ABB RobotStudio station: Solution_20200504-211433.rsstn

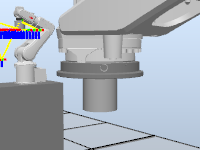
Station Solution (saved by RobotStudio 7.0.8743.626)
Controller Controller
  mechanical unit ROB_1: IRB120_3_58__01, 6 joints, base frame (-200, 0, 800) mm
  mechanical unit ROB_2: IRB120_3_58__01_2, 6 joints, base frame (200, 0, 800) mm, rotated rx 0 ry 0 rz 180 deg
  mechanical unit ROB_3: IRB760_450_318__01, 6 joints, base frame (0, 4000, 0) mm
Layout (positions relative to the parent item):
  - IRB120_3_58__01 [mechanism, from Robots\IRB120_3_58_G_01.rslib] at (-200, 0, 800) mm; joint values [0, -0.7948, 0.351, 0, 2.0145, 0] (rad or m)
  - IRB120_3_58__01_2 [mechanism, from Robots\IRB120_3_58_G_01.rslib] at (200, 0, 800) mm, rotated rx 0 ry 0 rz 180 deg; joint values [0, -0.7948, 0.351, 0, 2.0145, 0] (rad or m)
  - IRB760_450_318__01 [mechanism, from Robots\IRB760_450_318__01.rslib] at (0, 4000, 0) mm; joint values [-1.1097, -0.0075, 0.5664, -1.1097] (rad or m)
  - Part_1 [part]
  - Tool_1 [mechanism] at (-150, 0, 1400) mm, rotated rx 180 ry 0 rz 180 deg
      TCP Tool1 at (0, 0, 0) mm
      links: SimpleGripper
  - Tool_2 [mechanism] at (150, 0, 1400) mm, rotated rx 180 ry 0 rz 0 deg
      TCP Tool_2 at (0, 0, 0) mm
      links: SimpleGripper
  - Tool_3 [mechanism] at (765, 2460, 1100) mm, rotated rx 180 ry 0 rz 180 deg
      TCP Tool_3 at (0, 0, 0) mm
      links: SimpleGripper
Attachment: Tool_1 is attached to IRB120_3_58__01 / Link6
Attachment: Tool_2 is attached to IRB120_3_58__01_2 / Link6
Attachment: Tool_3 is attached to IRB760_450_318__01 / Link6
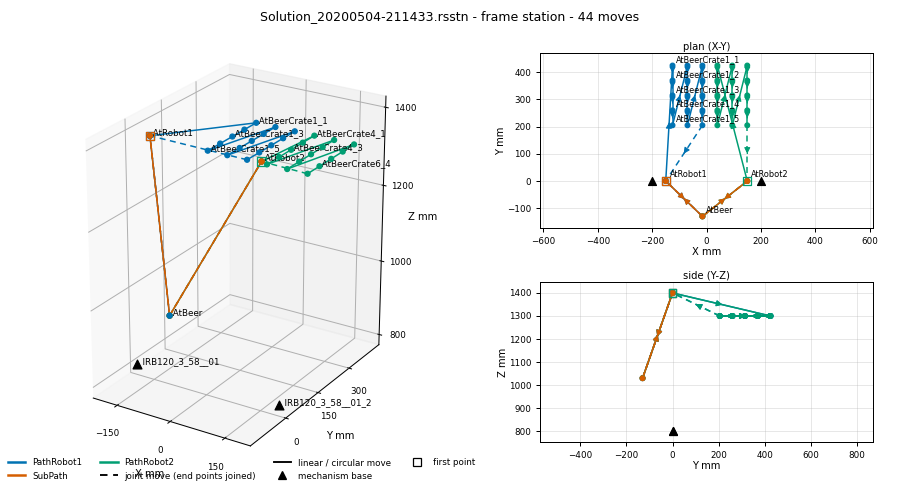
[picture p0: tool path of Solution_20200504-211433.rsstn in frame station, 44 of 44 moves have a stored position in this frame; points joined in program order, loops and branches not executed]
Targets, tools, work objects and paths stored in the station, written as RAPID:
! task T_ROB1
MODULE CalibData
  PERS tooldata Tool1:=[TRUE,[[0,0,0],[1,0,0,0]],[1,[0,0,1],[1,0,0,0],0,0,0]];
ENDMODULE

! task T_ROB1
MODULE Module1
  CONST robtarget AtBeer:=[[-15,-130,1030],[0,0,1,0],[-1,0,-1,0],[9E+09,9E+09,9E+09,9E+09,9E+09,9E+09]];
  CONST robtarget AtRobot1:=[[-150,0,1400],[0,0,1,0],[0,0,0,0],[9E+09,9E+09,9E+09,9E+09,9E+09,9E+09]];
  CONST robtarget AtBeerCrate1_1:=[[-125,425,1300],[0,0,1,0],[0,0,0,0],[9E+09,9E+09,9E+09,9E+09,9E+09,9E+09]];
  CONST robtarget AtBeerCrate1_2:=[[-125,370,1300],[0,0,1,0],[0,0,0,0],[9E+09,9E+09,9E+09,9E+09,9E+09,9E+09]];
  CONST robtarget AtBeerCrate1_3:=[[-125,315,1300],[0,0,1,0],[0,0,0,0],[9E+09,9E+09,9E+09,9E+09,9E+09,9E+09]];
  CONST robtarget AtBeerCrate1_4:=[[-125,260,1300],[0,0,1,0],[0,0,0,0],[9E+09,9E+09,9E+09,9E+09,9E+09,9E+09]];
  CONST robtarget AtBeerCrate1_5:=[[-125,205,1300],[0,0,1,0],[0,0,0,0],[9E+09,9E+09,9E+09,9E+09,9E+09,9E+09]];
  CONST robtarget AtBeerCrate2_1:=[[-70,425,1300],[0,0,1,0],[0,0,0,0],[9E+09,9E+09,9E+09,9E+09,9E+09,9E+09]];
  CONST robtarget AtBeerCrate2_2:=[[-70,370,1300],[0,0,1,0],[0,0,0,0],[9E+09,9E+09,9E+09,9E+09,9E+09,9E+09]];
  CONST robtarget AtBeerCrate2_3:=[[-70,315,1300],[0,0,1,0],[0,0,0,0],[9E+09,9E+09,9E+09,9E+09,9E+09,9E+09]];
  CONST robtarget AtBeerCrate2_4:=[[-70,260,1300],[0,0,1,0],[0,0,0,0],[9E+09,9E+09,9E+09,9E+09,9E+09,9E+09]];
  CONST robtarget AtBeerCrate2_5:=[[-70,205,1300],[0,0,1,0],[0,0,0,0],[9E+09,9E+09,9E+09,9E+09,9E+09,9E+09]];
  CONST robtarget AtBeerCrate3_1:=[[-15,425,1300],[0,0,1,0],[0,0,0,0],[9E+09,9E+09,9E+09,9E+09,9E+09,9E+09]];
  CONST robtarget AtBeerCrate3_2:=[[-15,370,1300],[0,0,1,0],[0,0,0,0],[9E+09,9E+09,9E+09,9E+09,9E+09,9E+09]];
  CONST robtarget AtBeerCrate3_3:=[[-15,315,1300],[0,0,1,0],[0,0,0,0],[9E+09,9E+09,9E+09,9E+09,9E+09,9E+09]];
  CONST robtarget AtBeerCrate3_4:=[[-15,260,1300],[0,0,1,0],[0,0,0,0],[9E+09,9E+09,9E+09,9E+09,9E+09,9E+09]];
  CONST robtarget AtBeerCrate3_5:=[[-15,205,1300],[0,0,1,0],[0,0,0,0],[9E+09,9E+09,9E+09,9E+09,9E+09,9E+09]];
  PROC main()
    PathRobot1;
  ENDPROC
  PROC PathRobot1()
    MoveJ AtRobot1,v2000,z100,Tool1\WObj:=wobj0;
    MoveL AtBeer,v2000,fine,Tool1\WObj:=wobj0;
    SetDO Do1Gripper,1;
    WaitTime 0.3;
    MoveJ AtRobot1,v2000,z100,Tool1\WObj:=wobj0;
    MoveL AtBeerCrate1_1,v2000,fine,Tool1\WObj:=wobj0;
    SubPath;
    MoveL AtBeerCrate1_2,v2000,fine,Tool1\WObj:=wobj0;
    SubPath;
    MoveL AtBeerCrate1_3,v2000,fine,Tool1\WObj:=wobj0;
    SubPath;
    MoveL AtBeerCrate1_4,v2000,fine,Tool1\WObj:=wobj0;
    SubPath;
    MoveL AtBeerCrate1_5,v2000,fine,Tool1\WObj:=wobj0;
    SubPath;
    MoveL AtBeerCrate2_1,v2000,fine,Tool1\WObj:=wobj0;
    SubPath;
    MoveL AtBeerCrate2_2,v2000,fine,Tool1\WObj:=wobj0;
    SubPath;
    MoveL AtBeerCrate2_3,v2000,fine,Tool1\WObj:=wobj0;
    SubPath;
    MoveL AtBeerCrate2_4,v2000,fine,Tool1\WObj:=wobj0;
    SubPath;
    MoveL AtBeerCrate2_5,v2000,fine,Tool1\WObj:=wobj0;
    SubPath;
    MoveL AtBeerCrate3_1,v2000,fine,Tool1\WObj:=wobj0;
    SubPath;
    MoveL AtBeerCrate3_2,v2000,fine,Tool1\WObj:=wobj0;
    SubPath;
    MoveL AtBeerCrate3_3,v2000,fine,Tool1\WObj:=wobj0;
    SubPath;
    MoveL AtBeerCrate3_4,v2000,fine,Tool1\WObj:=wobj0;
    SubPath;
    MoveL AtBeerCrate3_5,v2000,fine,Tool1\WObj:=wobj0;
    SetDO Do1Gripper,0;
    WaitTime 0.3;
    MoveJ AtRobot1,v2000,z100,Tool1\WObj:=wobj0;
  ENDPROC
  PROC SubPath()
    SetDO Do1Gripper,0;
    WaitTime 0.3;
    MoveJ AtRobot1,v2000,z100,Tool1\WObj:=wobj0;
    MoveL AtBeer,v2000,fine,Tool1\WObj:=wobj0;
    SetDO Do1Gripper,1;
    WaitTime 0.3;
    MoveJ AtRobot1,v2000,z100,Tool1\WObj:=wobj0;
  ENDPROC
ENDMODULE

! task T_ROB2
MODULE Module1
  CONST robtarget AtBeer:=[[-15,-130,1030],[0,1,0,0],[0,0,0,0],[9E+09,9E+09,9E+09,9E+09,9E+09,9E+09]];
  CONST robtarget AtRobot2:=[[150,0,1400],[0,1,0,0],[0,0,0,0],[9E+09,9E+09,9E+09,9E+09,9E+09,9E+09]];
  CONST robtarget AtBeerCrate4_1:=[[40,425,1300],[0,1,0,0],[-1,0,-1,0],[9E+09,9E+09,9E+09,9E+09,9E+09,9E+09]];
  CONST robtarget AtBeerCrate4_2:=[[40,370,1300],[0,1,0,0],[-1,0,-1,0],[9E+09,9E+09,9E+09,9E+09,9E+09,9E+09]];
  CONST robtarget AtBeerCrate4_3:=[[40,315,1300],[0,1,0,0],[-1,0,-1,0],[9E+09,9E+09,9E+09,9E+09,9E+09,9E+09]];
  CONST robtarget AtBeerCrate4_4:=[[40,260,1300],[0,1,0,0],[-1,0,-1,0],[9E+09,9E+09,9E+09,9E+09,9E+09,9E+09]];
  CONST robtarget AtBeerCrate4_5:=[[40,205,1300],[0,1,0,0],[-1,0,-1,0],[9E+09,9E+09,9E+09,9E+09,9E+09,9E+09]];
  CONST robtarget AtBeerCrate5_1:=[[95,425,1300],[0,1,0,0],[-1,0,-1,0],[9E+09,9E+09,9E+09,9E+09,9E+09,9E+09]];
  CONST robtarget AtBeerCrate5_2:=[[95,370,1300],[0,1,0,0],[-1,0,-1,0],[9E+09,9E+09,9E+09,9E+09,9E+09,9E+09]];
  CONST robtarget AtBeerCrate5_3:=[[95,315,1300],[0,1,0,0],[-1,0,-1,0],[9E+09,9E+09,9E+09,9E+09,9E+09,9E+09]];
  CONST robtarget AtBeerCrate5_4:=[[95,260,1300],[0,1,0,0],[-1,0,-1,0],[9E+09,9E+09,9E+09,9E+09,9E+09,9E+09]];
  CONST robtarget AtBeerCrate5_5:=[[95,205,1300],[0,1,0,0],[0,0,0,0],[9E+09,9E+09,9E+09,9E+09,9E+09,9E+09]];
  CONST robtarget AtBeerCrate6_1:=[[150,425,1300],[0,1,0,0],[0,0,0,0],[9E+09,9E+09,9E+09,9E+09,9E+09,9E+09]];
  CONST robtarget AtBeerCrate6_2:=[[150,370,1300],[0,1,0,0],[0,0,0,0],[9E+09,9E+09,9E+09,9E+09,9E+09,9E+09]];
  CONST robtarget AtBeerCrate6_3:=[[150,315,1300],[0,1,0,0],[0,0,0,0],[9E+09,9E+09,9E+09,9E+09,9E+09,9E+09]];
  CONST robtarget AtBeerCrate6_4:=[[150,260,1300],[0,1,0,0],[0,0,0,0],[9E+09,9E+09,9E+09,9E+09,9E+09,9E+09]];
  CONST robtarget AtBeerCrate6_5:=[[150,205,1300],[0,1,0,0],[0,0,0,0],[9E+09,9E+09,9E+09,9E+09,9E+09,9E+09]];
  PROC main()
    PathRobot2;
  ENDPROC
  PROC PathRobot2()
    MoveJ AtRobot2,v2000,z100,Tool2\WObj:=wobj0;
    WaitTime 1.5;
    MoveL AtBeer,v2000,fine,Tool2\WObj:=wobj0;
    SetDO Do2Gripper,0;
    WaitTime 0.3;
    MoveJ AtRobot2,v2000,z100,Tool2\WObj:=wobj0;
    MoveL AtBeerCrate4_1,v2000,fine,Tool2\WObj:=wobj0;
    SubPath;
    MoveL AtBeerCrate4_2,v2000,fine,Tool2\WObj:=wobj0;
    SubPath;
    MoveL AtBeerCrate4_3,v2000,fine,Tool2\WObj:=wobj0;
    SubPath;
    MoveL AtBeerCrate4_4,v2000,fine,Tool2\WObj:=wobj0;
    SubPath;
    MoveL AtBeerCrate4_5,v2000,fine,Tool2\WObj:=wobj0;
    SubPath;
    MoveL AtBeerCrate5_1,v2000,fine,Tool2\WObj:=wobj0;
    SubPath;
    MoveL AtBeerCrate5_2,v2000,fine,Tool2\WObj:=wobj0;
    SubPath;
    MoveL AtBeerCrate5_3,v2000,fine,Tool2\WObj:=wobj0;
    SubPath;
    MoveL AtBeerCrate5_4,v2000,fine,Tool2\WObj:=wobj0;
    SubPath;
    MoveL AtBeerCrate5_5,v2000,fine,Tool2\WObj:=wobj0;
    SubPath;
    MoveL AtBeerCrate6_1,v2000,fine,Tool2\WObj:=wobj0;
    SubPath;
    MoveL AtBeerCrate6_2,v2000,fine,Tool2\WObj:=wobj0;
    SubPath;
    MoveL AtBeerCrate6_3,v2000,fine,Tool2\WObj:=wobj0;
    SubPath;
    MoveL AtBeerCrate6_4,v2000,fine,Tool2\WObj:=wobj0;
    SubPath;
    MoveL AtBeerCrate6_5,v2000,fine,Tool2\WObj:=wobj0;
    SetDO Do2Gripper,0;
    WaitTime 0.3;
    MoveJ AtRobot2,v2000,z100,Tool2\WObj:=wobj0;
  ENDPROC
  PROC SubPath()
    SetDO Do2Gripper,0;
    WaitTime 0.3;
    MoveJ AtRobot2,v2000,z100,Tool2\WObj:=wobj0;
    MoveL AtBeer,v2000,fine,Tool2\WObj:=wobj0;
    SetDO Do2Gripper,1;
    WaitTime 0.3;
    MoveJ AtRobot2,v2000,z100,Tool2\WObj:=wobj0;
  ENDPROC
ENDMODULE

! task T_ROB2
MODULE CalibData
  PERS tooldata Tool2:=[TRUE,[[0,0,0],[1,0,0,0]],[1,[0,0,1],[1,0,0,0],0,0,0]];
  PERS tooldata Tool_2:=[TRUE,[[0,0,0],[1,0,0,0]],[1,[0,0,1],[1,0,0,0],0,0,0]];
ENDMODULE

! task T_ROB3
MODULE CalibData
  PERS tooldata Tool_3:=[TRUE,[[0,0,0],[1,0,0,0]],[1,[0,0,1],[1,0,0,0],0,0,0]];
ENDMODULE

! task T_ROB3
MODULE Module1
  CONST robtarget AtCrate:=[[765,2460,1100],[0,0,1,0],[0,0,0,0],[9E+09,9E+09,9E+09,9E+09,9E+09,9E+09]];
  CONST robtarget AtRobot3:=[[1000,3000,1500],[0,0,1,0],[0,0,0,0],[9E+09,9E+09,9E+09,9E+09,9E+09,9E+09]];
  CONST robtarget PAllet1_6:=[[1100,3500,400],[0,0.961261696,-0.275637356,0],[0,0,0,0],[9E+09,9E+09,9E+09,9E+09,9E+09,9E+09]];
  CONST robtarget Pallet1_5:=[[1370,3260,400],[0,0.961261696,-0.275637356,0],[0,0,0,0],[9E+09,9E+09,9E+09,9E+09,9E+09,9E+09]];
  CONST robtarget Pallet1_4:=[[1640,3050,400],[0,-0.48480962,0.874619707,0],[0,0,0,0],[9E+09,9E+09,9E+09,9E+09,9E+09,9E+09]];
  CONST robtarget Pallet1_1:=[[1860,3310,400],[0,0.961261696,-0.275637356,0],[0,0,0,0],[9E+09,9E+09,9E+09,9E+09,9E+09,9E+09]];
  CONST robtarget Pallet1_2:=[[1600,3550,400],[0,0.961261696,-0.275637356,0],[0,0,0,0],[9E+09,9E+09,9E+09,9E+09,9E+09,9E+09]];
  CONST robtarget Pallet1_3:=[[1340,3750,400],[0,-0.48480962,0.874619707,0],[0,0,0,0],[9E+09,9E+09,9E+09,9E+09,9E+09,9E+09]];
  CONST robtarget AboveCrate:=[[765,2460,1100],[0,0,1,0],[0,0,0,0],[9E+09,9E+09,9E+09,9E+09,9E+09,9E+09]];
ENDMODULE

